FUNCTION SUCCEEDED_AND_NOT_PENDING : BOOL
VAR_INPUT
	hr 	: DINT;
END_VAR
VAR
END_VAR

SUCCEEDED_AND_NOT_PENDING := hr >= 0 AND hr <> S_PENDING;

END_FUNCTION

(* stored: Version 1.1.0.1, ProductVersion 3.1.4026.18
   POU SUCCEEDED_AND_NOT_PENDING: Id {4a3707aa-19c7-47a8-892b-1feb62226184}, SpecialFunc None *)
